{attribute 'GeneratedUsingTerminal: KL1212'}
{attribute addProperty BoxType "KL1212"}
{attribute addProperty Id "InputAT %I*BOOL0ErrorAT %I*BOOL0PowerAT %Q*BOOL0"}
{attribute addProperty CRC "1927242550"}
{attribute addProperty Size "0"}
TYPE Channel_72DF6336 :
STRUCT
	{attribute addProperty Name "Input"}
	Input AT %I* : BOOL;
	{attribute addProperty Name "Error"}
	Error AT %I* : BOOL;
	{attribute addProperty Name "Power"}
	Power AT %Q* : BOOL;
END_STRUCT
END_TYPE

(* stored: Version 1.2.0.0, ProductVersion 3.1.4024.9
   DUT Channel_72DF6336: Id {6521725c-9c84-4efd-b3de-8f7342f8224c} *)
